// TIA Portal V19 export
TYPE "type_parameterError"
// stored: Access Published
   STRUCT
      cms : Array[0..99] of "type_cmParError";
      material { S7_SetPoint := 'True'} : Array[0..99] of "type_materialParError";
   END_STRUCT;
END_TYPE
